FUNCTION_BLOCK AS_SPLIT_SIGNED (* Teilt einen SINT-Wert in 2 einseitige Betragswerte auf (z.B. fuer 2 getrennte Bargraphen links/rechts einer Mittelstellung): NEG_MAG = MAX(0,-Y), POS_MAG = MAX(0,Y). Sonderfall Y=SINT#-128 (SINT-Minimum): -Y wuerde ueberlaufen (Zweierkomplement, |MIN| > MAX) - in diesem Fall wird NEG_MAG auf SINT#127 (SINT-Maximum) begrenzt (Regelungstechnik: Saettigung statt Ueberlauf/Vorzeichenwechsel). Adapter-Wrapper um SPLIT_SIGNED_SINT (reine Value/Event-Berechnung), Event je Seite nur bei tatsaechlicher Wertaenderung dank je einem E_D_FF_ANY (generischer Standardbaustein) pro Ausgang. *)
  (* Standard: 61499-2 *)
  (* Version 3.0, 2026-09-11, Franz Höpfinger, Vereinfacht: kombinatorische 3-Zustands-ECC (EMIT_BOTH/EMIT_NEG_ONLY/EMIT_POS_ONLY) durch Composite-FB ersetzt - reine Berechnung jetzt in SPLIT_SIGNED_SINT (Value/Event), Event-Dedup je Seite durch je einen generischen E_D_FF_ANY *)
  (* Version 2.3, 2026-09-11, Franz Höpfinger, Alle Literale vollqualifiziert (SINT#...) statt unqualifizierter Zahlenliterale *)
  (* Version 2.2, 2026-09-11, Franz Höpfinger, Ueberlauf bei Y=SINT#-128 (SINT-Minimum) abgefangen: -Y waere nicht als SINT darstellbar (|MIN|>MAX bei Zweierkomplement) - NEG_MAG saettigt in diesem Fall auf SINT#127 statt zu ueberlaufen *)
  (* Version 2.1, 2026-09-11, Franz Höpfinger, Kein eigener prevNeg/prevPos-Internal mehr noetig - Vergleich direkt gegen NEG_MAG.D1/POS_MAG.D1 (Plug-Ausgang haelt den letzten Wert bereits selbst) *)
  (* Version 2.0, 2026-09-11, Franz Höpfinger, Event nur noch bei tatsaechlicher Wertaenderung je Seite (vorher: bei jedem Y-Update immer beide Events, unabhaengig ob sich der Wert aendert) *)
  (* Version 1.0, 2026-09-11, Franz Höpfinger, Typfamilie zu AR_SPLIT_SIGNED, generisch fuer jede aehnliche Anzeige *)
  PACKAGE adapter::Engineering::splitting::signed;
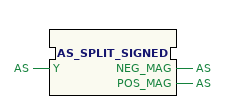
  SOCKETS
    Y : adapter::types::unidirectional::AS; (* Eingangswert *)
  END_SOCKETS
  PLUGS
    NEG_MAG : adapter::types::unidirectional::AS; (* MAX(0, -Y) - Betrag der negativen Auslenkung, bei Y=SINT#-128 gesaettigt auf SINT#127, Event nur bei Aenderung *)
    POS_MAG : adapter::types::unidirectional::AS; (* MAX(0, Y) - Betrag der positiven Auslenkung, Event nur bei Aenderung *)
  END_PLUGS
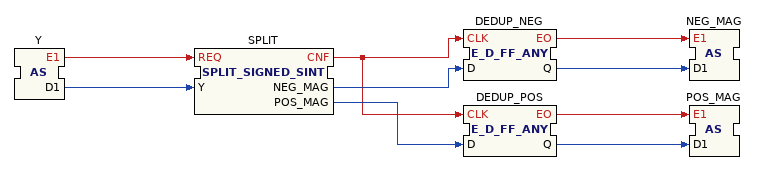
  FBS
    SPLIT : adapter::Engineering::splitting::signed::SPLIT_SIGNED_SINT;
    DEDUP_NEG : iec61499::events::E_D_FF_ANY;
    DEDUP_POS : iec61499::events::E_D_FF_ANY;
  END_FBS
  EVENT_CONNECTIONS
    Y.E1 TO SPLIT.REQ;
    SPLIT.CNF TO DEDUP_NEG.CLK;
    SPLIT.CNF TO DEDUP_POS.CLK;
    DEDUP_NEG.EO TO NEG_MAG.E1;
    DEDUP_POS.EO TO POS_MAG.E1;
  END_CONNECTIONS
  DATA_CONNECTIONS
    Y.D1 TO SPLIT.Y;
    SPLIT.NEG_MAG TO DEDUP_NEG.D;
    SPLIT.POS_MAG TO DEDUP_POS.D;
    DEDUP_NEG.Q TO NEG_MAG.D1;
    DEDUP_POS.Q TO POS_MAG.D1;
  END_CONNECTIONS
END_FUNCTION_BLOCK
